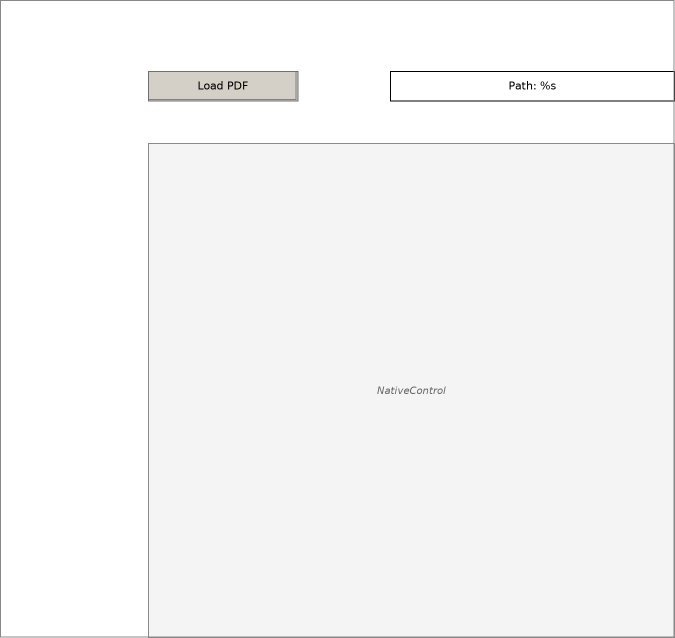
VISUALIZATION Visualization  // 675x638
    NativeControl (148,143 527x495)
        Calls[0]: Method=LoadFile, Variable=MAIN.bLoad
        Parameters[0]: Var=MAIN.sPath
        p3873840581: AcroPDF.PDF.1
    Button (148,71 150x30), "Load PDF"
        tap MAIN.bLoad
    Rectangle (390,71 285x30), "Path: %s", text variable: MAIN.sPath
END_VISUALIZATION

(* stored: Version 1.1.0.1, ProductVersion 3.1.4024.3
   Visu Visualization: Id {3c383d8a-9ab7-48be-a31a-2853fedd5e93} *)
